INTERFACE I_CustomMode EXTENDS I_PackMLMode

END_INTERFACE

(* stored: Version 1.1.0.1, ProductVersion 3.1.4024.12
   Itf I_CustomMode: Id {54875696-6434-4991-bcbd-4134edd74cd8} *)
